# EPICS autosave request: iocs/roperIOC/iocBoot/iocRoper/auto_settings.req
file "roper_settings.req",        P=$(P),  R=cam1:
file "NDStdArrays_settings.req",  P=$(P),  R=image1:
file "commonPlugin_settings.req", P=$(P)
